FUNCTION_BLOCK PickNPlace (* Template for an empty basic function block *)
  (* Standard: 61499-2 *)
  (* Version 1.0, 2018-09-13, az *)
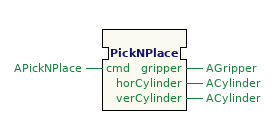
  SOCKETS
    cmd : APickNPlace;
  END_SOCKETS
  PLUGS
    gripper : AGripper;
    horCylinder : ACylinder;
    verCylinder : ACylinder;
  END_PLUGS
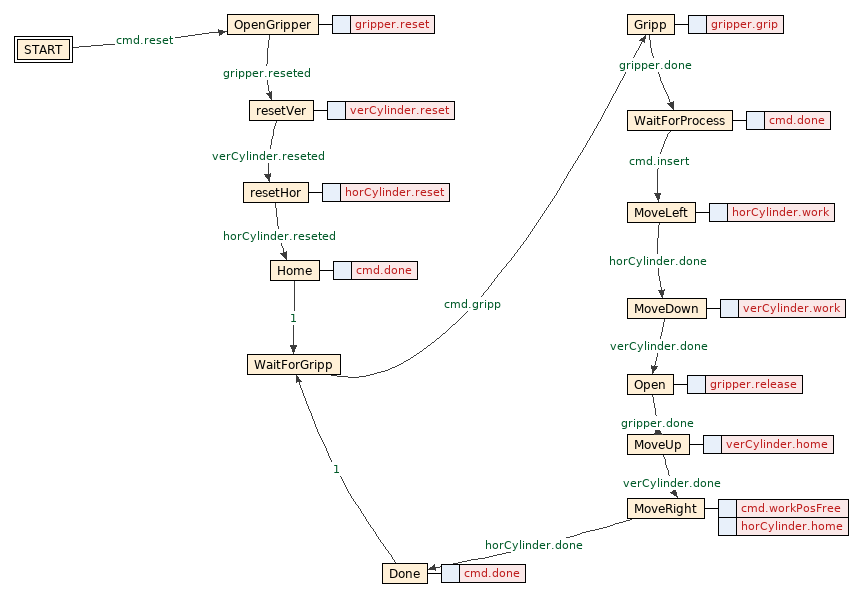
  EC_STATES
    START; (* Initial State *)
    OpenGripper : -> gripper.reset;
    resetVer : -> verCylinder.reset;
    resetHor : -> horCylinder.reset;
    Home : -> cmd.done;
    WaitForGripp;
    Gripp : -> gripper.grip;
    WaitForProcess : -> cmd.done;
    MoveLeft : -> horCylinder.work;
    MoveDown : -> verCylinder.work;
    Open : -> gripper.release;
    MoveUp : -> verCylinder.home;
    MoveRight : -> cmd.workPosFree, -> horCylinder.home;
    Done : -> cmd.done;
  END_STATES
  EC_TRANSITIONS
    START TO OpenGripper := cmd.reset;
    OpenGripper TO resetVer := gripper.reseted;
    resetVer TO resetHor := verCylinder.reseted;
    resetHor TO Home := horCylinder.reseted;
    Home TO WaitForGripp := 1;
    Done TO WaitForGripp := 1;
    WaitForGripp TO Gripp := cmd.gripp;
    Gripp TO WaitForProcess := gripper.done;
    WaitForProcess TO MoveLeft := cmd.insert;
    MoveLeft TO MoveDown := horCylinder.done;
    MoveDown TO Open := verCylinder.done;
    Open TO MoveUp := gripper.done;
    MoveUp TO MoveRight := verCylinder.done;
    MoveRight TO Done := horCylinder.done;
  END_TRANSITIONS
END_FUNCTION_BLOCK
